FUNCTION_BLOCK M3RotationGoto EXTENDS BaseProcess
VAR_INPUT
	///Arguments to be set, before writing do_request TRUE
	{attribute 'OPC.UA.DA' := '1'}
	set: M3RotationGotoArgs;
END_VAR
VAR_OUTPUT
	///Arguments in use by the process, if do_request was accepted
	{attribute 'OPC.UA.DA' := '1'}
	{attribute 'OPC.UA.DA.Access' := '1'}
	get: M3RotationGotoArgs;
END_VAR
VAR_IN_OUT
END_VAR
VAR
END_VAR

IF do_request THEN
    do_request_result := request(
    position := set.position,
    offset := set.offset);
    do_request := FALSE;
END_IF;
SUPER^();

{attribute 'TcRpcEnable' := '1'}
METHOD start
VAR_INPUT
	///Position setpoint of the rotation stage, in degrees
	position: LREAL;
	///Offset setpoint between the motors of the rotation stage, in degrees
	offset: LREAL;
END_VAR
VAR_OUTPUT
END_VAR
VAR_IN_OUT
END_VAR
VAR
END_VAR
THIS^.get.position := position;
THIS^.get.offset := offset;
THIS^.statuses.busyStatus( isBusy := TRUE );
THIS^.statuses.healthStatus( isGood := TRUE );
END_METHOD

{attribute 'TcRpcEnable' := '1'}
METHOD request : RequestResults
VAR_INPUT
	///Position setpoint of the rotation stage, in degrees
	position: LREAL;
	///Offset setpoint between the motors of the rotation stage, in degrees
	offset: LREAL;
END_VAR
VAR_OUTPUT
END_VAR
VAR_IN_OUT
END_VAR
VAR
END_VAR
IF THIS^.statuses.enabledStatus.enabled THEN
    THIS^.start(
        position := position,
        offset := offset);
    request := RequestResults.ACCEPTED;
ELSE
    request := RequestResults.REJECTED;
END_IF;
END_METHOD

END_FUNCTION_BLOCK

(* stored: Version 1.1.0.1, ProductVersion 3.1.4019.2
   POU M3RotationGoto: Id {cc0ad3ce-5966-4307-aa2d-89b3b10fd304}, SpecialFunc None
   Method start: Id {afe792d6-0db4-41dc-94e8-a776609af7d1}
   Method request: Id {b2c2619d-83ce-4342-b6fe-94b7452308e6} *)
